// TIA Portal V18 export
VAR_GLOBAL   // PLC tag table "Default tag table"
   D_INPUT AT %I0.0 : "DI";
   A_IN AT %I100.0 : "AI";
   RTD_IN AT %I108.0 : "RTD";
   D_OUTPUT AT %Q0.0 : "DO";
   A_OUT AT %Q100.0 : "AO";
   System_Byte AT %MB1 : Byte;
   FirstScan AT %M1.0 : Bool;
   DiagStatusUpdate AT %M1.1 : Bool;
   AlwaysTRUE AT %M1.2 : Bool;
   AlwaysFALSE AT %M1.3 : Bool;
   Clock_Byte AT %MB0 : Byte;
   Clock_10Hz AT %M0.0 : Bool;
   Clock_5Hz AT %M0.1 : Bool;
   "Clock_2.5Hz" AT %M0.2 : Bool;
   Clock_2Hz AT %M0.3 : Bool;
   "Clock_1.25Hz" AT %M0.4 : Bool;
   Clock_1Hz AT %M0.5 : Bool;
   "Clock_0.625Hz" AT %M0.6 : Bool;
   "Clock_0.5Hz" AT %M0.7 : Bool;
   Tag_1 AT %M5.0 : Bool;
   Tag_2 AT %M55.0 : Bool;
   Tag_3 AT %M75.0 : Bool;
END_VAR
VAR_GLOBAL CONSTANT   // user constants
   "None(2)" : Pip := 65535;
   "Automatic update(2)" : Pip := 0;
   "PIP 1(2)" : Pip := 1;
   "PIP 2(2)" : Pip := 2;
   "PIP 3(2)" : Pip := 3;
   "PIP 4(2)" : Pip := 4;
   "PIP 5" : Pip := 5;
   "PIP 6" : Pip := 6;
   "PIP 7" : Pip := 7;
   "PIP 8" : Pip := 8;
   "PIP 9" : Pip := 9;
   "PIP 10" : Pip := 10;
   "PIP 11" : Pip := 11;
   "PIP 12" : Pip := 12;
   "PIP 13" : Pip := 13;
   "PIP 14" : Pip := 14;
   "PIP 15" : Pip := 15;
   "PIP 16" : Pip := 16;
   "PIP 17" : Pip := 17;
   "PIP 18" : Pip := 18;
   "PIP 19" : Pip := 19;
   "PIP 20" : Pip := 20;
   "PIP 21" : Pip := 21;
   "PIP 22" : Pip := 22;
   "PIP 23" : Pip := 23;
   "PIP 24" : Pip := 24;
   "PIP 25" : Pip := 25;
   "PIP 26" : Pip := 26;
   "PIP 27" : Pip := 27;
   "PIP 28" : Pip := 28;
   "PIP 29" : Pip := 29;
   "PIP 30" : Pip := 30;
   "PIP 31" : Pip := 31;
   "PIP OB Servo(2)" : Pip := 32768;
   "Local~MC(2)" : Hw_SubModule := 51;
   "Local~Common(2)" : Hw_SubModule := 50;
   "Local~Device(2)" : Hw_Device := 32;
   "Local~Configuration(2)" : Hw_SubModule := 33;
   "Local~Display" : Hw_SubModule := 54;
   "Local~Exec(2)" : Hw_SubModule := 52;
   "Local(2)" : Hw_SubModule := 49;
   "Local~PROFINET_interface_1(2)" : Hw_Interface := 64;
   "Local~PROFINET_interface_1~Port_1(2)" : Hw_Interface := 65;
   "Local~PROFINET_interface_1~Port_2" : Hw_Interface := 66;
   "Local~Virtual_communication_interface" : Hw_Interface := 135;
   "Local~License_Manager" : Hw_SubModule := 42;
   "OB_Main(2)" : OB_PCYCLE := 1;
END_VAR
